# EPICS autosave request: iocBoot/sioc-cha-bkhM2/bkh2.req
file ../bkhMot.req P=$(P),MOT=2531-1,M=$(M)
file ../bkhMot.req P=$(P),MOT=2531-2,M=$(M)

$(P):AI:3132-$(M):CH1.DESC
$(P):AO:3132-$(M):CH1:A
$(P):AO:3132-$(M):CH1:B

$(P):AI:3132-$(M):CH2.DESC
$(P):AO:3132-$(M):CH2:A
$(P):AO:3132-$(M):CH2:B

$(P):AO:4132-$(M):CH1.DESC
$(P):AO:4132-$(M):CH1

$(P):AO:4132-$(M):CH2.DESC
$(P):AO:4132-$(M):CH2
